// TIA Portal V20 export
// export: Created 2025-12-01T14:57:18.0850815Z, ExportSetting None, DisplayName Totally Integrated Automation Portal, DisplayVersion V20 Update 3, DisplayName TIA Portal Openness, DisplayVersion V20 Update 3, DisplayName TIA Portal Version Control Interface, DisplayVersion V20 Update 3, DisplayName STEP 7 Professional, DisplayVersion V20 Update 3, DisplayName STEP 7 Safety, DisplayVersion V20 Update 2, DisplayName WinCC Basic/Comfort/Advanced, DisplayVersion V20 Update 3, DisplayName WinCC Professional, DisplayVersion V20 Update 3, DisplayName WinCC Unified, DisplayVersion V20 Update 3
DATA_BLOCK "DB905_Estado_Escaners"   // DB905
{ S7_Optimized_Access := 'FALSE' }
// stored: AutoNumber false
   VAR
      total_registros : UInt;
      long_registro : Int := 50;
      offset_primero : Int := 6;
      Escaner { S7_SetPoint := 'True'} : Array[1.."ROUT_Max_Scanners"] of "ROUT_Datos_Pantalla_Scanner";   // Variable comodín provisional
   END_VAR
BEGIN
END_DATA_BLOCK
